TYPE ST_RxHmi :
STRUCT
	counter : UDINT := 0;
	winchJogUp : BOOL;
	winchJogDown : BOOL;
	xboxLeftX : REAL;
	xboxLeftY : REAL;
	xboxRightX : REAL;
	xboxRightY : REAL;
	xboxLT : REAL;
	xboxRT : REAL;
END_STRUCT
END_TYPE

(* stored: Version 1.1.0.1, ProductVersion 3.1.4022.7
   DUT ST_RxHmi: Id {896c6bcd-7067-44e9-b168-de4b21e4463e} *)
